// TwinCAT 3 PLC project MAS418_PLC
// ProgramVersion: 3.1.4023.0
// libraries:
//   Tc2_Standard, * (Beckhoff Automation GmbH)
//   Tc2_System, * (Beckhoff Automation GmbH)
//   Tc3_Module, * (Beckhoff Automation GmbH)
// project tree:
//   DUTs/ E_ControlBox.TcDUT, E_Mode.TcDUT, E_Status.TcDUT, ST_Joystick.TcDUT, ST_JoystickInputScaling.TcDUT, ST_Params.TcDUT, ST_Position.TcDUT, ST_PressureSensors.TcDUT, ST_ValveDeadBand.TcDUT
//   Fbs/ FB_ControlBox.TcPOU, FB_Encoder.TcPOU, FB_JoystickInputScaling.TcPOU, FB_RealControlBox_.TcPOU, FB_12bIntToReal.TcPOU, FB_ValveOutput.TcPOU, FB_VirtualControlBox.TcPOU
//   / GlobalTextList.TcGTLO, I_ControlBox.TcIO, I_Crane.TcIO, PlcTask.TcTTO, Visualization Manager.TcVMO (not stored)
//   GVLs/ CONSTANTS.TcGVL, INPUT.TcGVL, OUTPUTS.TcGVL, ScaledInputs.TcGVL, VirtualControlBox.TcGVL, Working.TcGVL
//   POUs/ CraneControl.TcPOU, FU_Scale_IO.TcPOU, MAIN.TcPOU
//   VISUs/ VirtualControlBox.TcVIS
// real-time tasks:
//   TASK PlcTask: cycle T#10ms, priority 20, ADS port 350
// I/O:
//   DEVICE Device 2 (EtherCAT), AmsNetId 5.80.90.242.3.1
//     Term 1 (EK1200) [EK1200-5000 EtherCAT Power supply (2A E-Bus)]
//       Term 10 (EL2008-0015) [EL2008-0015 8Ch. Dig. Output 24V DC, 0.35A, not short-circuit proof]
//       Term 3 (EL9011) [EL9011 End Terminal]
//   DEVICE Device 5 (EtherCAT), AmsNetId 5.80.90.242.6.1
//     Term 12 (EK1100) [EK1100 EtherCAT Coupler (2A E-Bus)]
//       DI1(EL1008) [EL1008 8Ch. Dig. Input 24V, 3ms]
//       DO1(EL2008) [EL2008 8Ch. Dig. Output 24V, 0.5A]
//       AI1(EL3068) [EL3068 8Ch. Ana. Input 0-10V]
//       AI2(EL3068) [EL3068 8Ch. Ana. Input 0-10V]
//       AI3(EL3174) [EL3174 4Ch. Ana. Input +/-10V Diff., +/-20mA SingleEnded, 16 Bit]
//       AI4(EL3255) [EL3255 5Ch. potentiometer measurement with sensor supply]
//       Term 19 (EL4104) [EL4104 4Ch. Ana. Output 0-10V, 16bit]
//       AO1(EL9011) [EL9011 End Terminal]
//     Box 20 (Fraba EtherCAT) [Absolute Rotary Encoder IXARC V01.05]
// variable links:
//   MAS418-PLC Instance <-> Device 5 (EtherCAT)/Box 20 (Fraba EtherCAT)
//     PlcTask Inputs/INPUT.nEncoder <-> Encoder/Position Value
//   MAS418-PLC Instance <-> Device 5 (EtherCAT)/Term 12 (EK1100)/AI1(EL3068)
//     PlcTask Inputs/INPUT.nPC_A <-> AI Standard Channel 4/Value
//     PlcTask Inputs/INPUT.nPC_B <-> AI Standard Channel 3/Value
//     PlcTask Inputs/INPUT.nPR <-> AI Standard Channel 2/Value
//     PlcTask Inputs/INPUT.nPS <-> AI Standard Channel 1/Value
//     PlcTask Inputs/INPUT.nPW_A <-> AI Standard Channel 7/Status
//     PlcTask Inputs/INPUT.nPW_A1 <-> AI Standard Channel 5/Value
//     PlcTask Inputs/INPUT.nPW_B <-> AI Standard Channel 8/Value
//     PlcTask Inputs/INPUT.nPW_B1 <-> AI Standard Channel 6/Value
//   MAS418-PLC Instance <-> Device 5 (EtherCAT)/Term 12 (EK1100)/AI2(EL3068)
//     PlcTask Inputs/INPUT.nPW_D <-> AI Standard Channel 1/Value
//     PlcTask Inputs/INPUT.nQW <-> AI Standard Channel 2/Value
//   MAS418-PLC Instance <-> Device 5 (EtherCAT)/Term 12 (EK1100)/AI4(EL3255)
//     PlcTask Inputs/INPUT.nJoyX <-> AI Standard Channel 2/Value
//     PlcTask Inputs/INPUT.nJoyY <-> AI Standard Channel 3/Value
//     PlcTask Inputs/INPUT.nXc <-> AI Standard Channel 1/Value
//   MAS418-PLC Instance <-> Device 5 (EtherCAT)/Term 12 (EK1100)/DI1(EL1008)
//     PlcTask Inputs/INPUT.bAuto <-> Channel 2/Input
//     PlcTask Inputs/INPUT.bJoystick <-> Channel 5/Input
//     PlcTask Inputs/INPUT.bManual <-> Channel 1/Input
//     PlcTask Inputs/INPUT.bStart <-> Channel 3/Input
//     PlcTask Inputs/INPUT.bStop <-> Channel 4/Input
//   MAS418-PLC Instance <-> Device 5 (EtherCAT)/Term 12 (EK1100)/DO1(EL2008)
//     PlcTask Outputs/OUTPUTS.bEnableCylValve <-> Channel 4/Output
//     PlcTask Outputs/OUTPUTS.bEnableWinchValve <-> Channel 3/Output
//     PlcTask Outputs/OUTPUTS.bGreenLed <-> Channel 1/Output
//     PlcTask Outputs/OUTPUTS.bRedLed <-> Channel 2/Output
//   MAS418-PLC Instance <-> Device 5 (EtherCAT)/Term 12 (EK1100)/Term 19 (EL4104)
//     PlcTask Outputs/OUTPUTS.nCylValveOut <-> AO Output Channel 2/Analog output
//     PlcTask Outputs/OUTPUTS.nWinchValveOut <-> AO Output Channel 1/Analog output

CONFIGURATION MAS418_PLC
    RESOURCE PLC ON TwinCAT3
        TASK PlcTask(INTERVAL := T#10ms, PRIORITY := 20);
        PROGRAM MAIN WITH PlcTask : MAIN;
    END_RESOURCE
END_CONFIGURATION

// ---- DUTs/E_ControlBox.TcDUT
{attribute 'qualified_only'}
{attribute 'strict'}
TYPE E_ControlBox :
(
	VirtualControlBox,
	RealControlBox
);
END_TYPE

// ---- DUTs/E_Mode.TcDUT
{attribute 'qualified_only'}
{attribute 'strict'}
TYPE E_Mode :
(
	AUTO := 0,
	OFF := 1,
	MANUAL := 2
);
END_TYPE

// ---- DUTs/E_Status.TcDUT
{attribute 'qualified_only'}
{attribute 'strict'}
TYPE E_Status :
(
	NotReady,
	Ready,
	Starting,
	Running,
	Stopping,
	Fault,
	Joystick
);
END_TYPE

// ---- DUTs/ST_Joystick.TcDUT
TYPE ST_Joystick :
STRUCT
	X : LREAL;
	Y : LREAL;
	Topswitch : BOOL;
END_STRUCT
END_TYPE

// ---- DUTs/ST_JoystickInputScaling.TcDUT
TYPE ST_JoystickInputScaling :
STRUCT
	
    fMaxInputValue : LREAL := 20509.0;
    fMinInputValue : LREAL := 11787.0;
    fNeutralInputValue : LREAL := 16175;
    fNeutralDeadband : LREAL := 50.0;
    fMaxOutputValue : LREAL := 1.0;
    fMinOutputValue : LREAL := -1.0;
    fNeutralOutputValue : LREAL := 0.0;

END_STRUCT
END_TYPE

// ---- DUTs/ST_Params.TcDUT
TYPE ST_Params :
STRUCT
	fEncoderOffset : LREAL;
END_STRUCT
END_TYPE

// ---- DUTs/ST_Position.TcDUT
TYPE ST_Position :
STRUCT
	winch : REAL;
	cylinder : REAL;
END_STRUCT
END_TYPE

// ---- DUTs/ST_PressureSensors.TcDUT
TYPE ST_PressureSensors :
STRUCT
	SupplyPres : REAL;
	ReturnPres : REAL;
	CylPistSide : REAL;
	CylRodSide : REAL;
	WinchInlet : REAL;
	WinchInlet2 : REAL;
	WinchOutlet : REAL;
	WinchOutlet2 : REAL;
	WinchDrain : REAL;
END_STRUCT
END_TYPE

// ---- DUTs/ST_ValveDeadBand.TcDUT
TYPE ST_ValveDeadBand :
STRUCT
	
    fPosMax : LREAL := 29490.0;
    fPosMin : LREAL  := 20950.0;
    fNegMin : LREAL  := 18250.0;
    fNegMax : LREAL  := 9830.0;

END_STRUCT
END_TYPE

// ---- GVLs/CONSTANTS.TcGVL
{attribute 'qualified_only'}
VAR_GLOBAL
	fDrumD : REAL := 0.475; //m
	fGearRatio : REAL := 1/20;
	//fMdisplacement	: REAL := 
	
END_VAR

// ---- GVLs/INPUT.TcGVL
{attribute 'qualified_only'}
VAR_GLOBAL
//	nJoyXRaw : INT;
//	nJoyYRaw : INT;
//	bJoySW 	: BOOL;
	
	//Digital
	bManual AT %I*: BOOL;
	bAuto AT %I*: BOOL;
	bStart AT %I*: BOOL;
	bStop AT %I*: BOOL;
	bJoystick AT %I*: BOOL;
	
	//Encoder
	nEncoder AT %I*: UDINT;
	
	//Analog Flow/pressure
	nPS AT %I*: INT;
	nPR AT %I*: INT;
	nPC_B  AT %I*: INT;
	nPC_A  AT %I*: INT;
	nPW_A1  AT %I*: INT;
	nPW_B1 AT %I*: INT;
	nPW_A AT %I*: INT;
	nPW_B AT %I*: INT;
	nPW_D AT %I*: INT;
	nQW AT %I*: INT;
	
	//Analog 
	nXc AT %I*: INT;
	//nJoy
	nJoyX AT %I*: INT;
	nJoyY AT %I*: INT;
	
//	fCylinderPositionSensor : REAL;
//	fWinchEncodder : REAL;
//	stPressureSensors : ST_PressureSensors;
//	WinchInletFlow : REAL;
	//I
END_VAR

// ---- GVLs/OUTPUTS.TcGVL
{attribute 'qualified_only'}
VAR_GLOBAL
	//bLightRed : BOOL := FALSE;
	//bLightGreen : BOOL := FALSE;
	//CylinderValve : REAL := 0; //initial value
	//WinchValve : REAL := 0; //initial value
	
	//Digital
	bGreenLed AT %Q*: BOOL;
	bRedLed AT %Q*: BOOL;
	bEnableWinchValve AT %Q*: BOOL;
	bEnableCylValve AT %Q*: BOOL;
	
	//Analog
	nWinchValveOut AT %Q*: INT;
	nCylValveOut AT %Q*: INT;
	
END_VAR

// ---- GVLs/ScaledInputs.TcGVL
{attribute 'qualified_only'}
VAR_GLOBAL
	stJoystick : ST_Joystick;
	
	//Analog Flow/pressure
	fPS : LREAL;
	fPR : LREAL;
	fPC_B : LREAL;
	fPC_A : LREAL;
	fPW_A1 : LREAL;
	fPW_B1 : LREAL;
	fPW_A : LREAL;
	fPW_B : LREAL;
	fPW_D : LREAL;
	fQW : LREAL;
	fXc: LREAL;
	
	fEncoder : LREAL;
	
	
	
END_VAR

// ---- GVLs/VirtualControlBox.TcGVL
{attribute 'qualified_only'}
VAR_GLOBAL
	bSTOP : BOOL := FALSE;
	bSTART : BOOL := FALSE;
	//bLightRed : BOOL := FALSE;
	//bLightGreen : BOOL := FALSE;
	bAuto : BOOL;
	bManual : BOOL;
	stJOY : ST_Joystick;
	//eMode : E_Mode;// := E_Mode.OFF;
	//strMode : STRING;
	//strStatus : STRING;
	//eStatus : E_Status;// := E_Status.NotReady;
	//eMode : E_Mode;// := E_Mode.OFF;
END_VAR

// ---- GVLs/Working.TcGVL
{attribute 'qualified_only'}
VAR_GLOBAL
	eMode : E_Mode;
	eStatus : E_Status := E_Status.NotReady; //Initial status
	strMode : STRING;
	strStatus : STRING;
END_VAR

// ---- I_ControlBox.TcIO
INTERFACE I_ControlBox

METHOD Joystick
VAR_INPUT
	//stJoystick : ST_Joystick;
END_VAR
VAR_OUTPUT
	stJoystick : ST_Joystick;
END_VAR
END_METHOD

METHOD Mode
VAR_INPUT
	//bAuto : BOOL;
	//bManual : BOOL;
	//eMode	: E_Mode; //should I read this value Directly from the VirtualControlBox?
END_VAR
VAR_OUTPUT
	eMode : E_Mode;
END_VAR
END_METHOD

METHOD Status
VAR_INPUT
	//eMode	: E_Mode;
	//bStart	: BOOL;
	//bStop	: BOOL;
END_VAR
VAR_OUTPUT
	//eStatus : E_Status := E_Status.NotReady;
END_VAR
END_METHOD

END_INTERFACE

// ---- I_Crane.TcIO
INTERFACE I_Crane

METHOD ControlValveOutput
VAR_INPUT
END_VAR
END_METHOD

METHOD FLOW : REAL
VAR_INPUT
END_VAR
END_METHOD

METHOD Position : ST_Position
VAR_INPUT
END_VAR
END_METHOD

METHOD Pressure : REAL
VAR_INPUT
END_VAR
END_METHOD

END_INTERFACE

// ---- POUs/MAIN.TcPOU
PROGRAM MAIN
VAR
END_VAR

CraneControl();

END_PROGRAM

// ---- POUs/CraneControl.TcPOU
PROGRAM CraneControl
VAR
	fbControlBox : FB_ControlBox;
	fbScaleOutputs : FB_ValveOutput;
	stValveDeadband : ST_ValveDeadBand;
	//eMode : E_Mode;
	eStatus : E_Status;
	bEnableCylinder : BOOL;
	bEnableWinch	: BOOL;
END_VAR

fbControlBox(eControlBox := E_ControlBox.VirtualControlBox); // set to true to use real controlbox

FU_Scale_IO();

eStatus:=Working.eStatus;
//Control Lights
IF eStatus = E_Status.Running THEN
	OUTPUTS.bGreenLed := TRUE;
	bEnableCylinder := TRUE;
	IF ScaledInputs.stJoystick.Topswitch THEN
		bEnableWinch := TRUE;
	ELSE
		bEnableWinch := FALSE;
	END_IF
ELSE
	OUTPUTS.bGreenLed := FALSE;
	bEnableCylinder := FALSE;
	bEnableWinch := FALSE;
END_IF

IF eStatus = E_Status.Stopping OR eStatus = E_Status.Fault THEN
	OUTPUTS.bRedLed := TRUE;
ELSE
	OUTPUTS.bRedLed := FALSE;
END_IF


//Outputs
fbScaleOutputs(bEnable:=bEnableCylinder, 
			bDeadBandCompOn:=TRUE, 
			stValveDeadBand:=stValveDeadband, 
			fNormalizedInput:=ScaledInputs.stJoystick.X, 
			bEnableValveOutput=>OUTPUTS.bEnableCylValve, 
			nOutput=>OUTPUTS.nCylValveOut);
			
fbScaleOutputs(bEnable:=bEnableWinch, 
			bDeadBandCompOn:=TRUE, 
			stValveDeadBand:=stValveDeadband, 
			fNormalizedInput:=ScaledInputs.stJoystick.Y, 
			bEnableValveOutput=>OUTPUTS.bEnableWinchValve, 
			nOutput=>OUTPUTS.nWinchValveOut);

END_PROGRAM

// ---- Fbs/FB_ControlBox.TcPOU
FUNCTION_BLOCK FB_ControlBox
VAR_INPUT
	eControlBox : E_ControlBox;
END_VAR
VAR
	fbVirtualControlBox : FB_VirtualControlBox;
	fbRealControlBox : FB_RealControlBox_;
	fbControlBox : I_ControlBox := fbVirtualControlBox; //Initial value
END_VAR

CASE eControlBox OF
	E_ControlBox.RealControlBox:
		fbControlBox := fbRealControlBox;
		
	E_ControlBox.VirtualControlBox:
		fbControlBox := fbVirtualControlBox;
END_CASE

fbControlBox.Mode();
fbControlBox.Status();
fbControlBox.Joystick();

END_FUNCTION_BLOCK

// ---- Fbs/FB_VirtualControlBox.TcPOU
FUNCTION_BLOCK FB_VirtualControlBox IMPLEMENTS I_ControlBox
VAR_INPUT
END_VAR
VAR_OUTPUT
END_VAR
VAR
END_VAR

//fbControlBox.Mode(
//	bAuto := VirtualControlBox.bAuto, 
//	bManual := VirtualControlBox.bManual,
//	eMode => VirtualControlBox.eMode
//);

//fbControlBox.Status(
//	eMode := VirtualControlBox.eMode,
//	bStart := VirtualControlBox.bSTART,
//	bStop := VirtualControlBox.bSTOP,
//	eStatus => VirtualControlBox.eStatus
//	);

{warning 'add method implementation '}
METHOD Joystick
VAR_INPUT
	//stJoystick	: ST_Joystick;
END_VAR
VAR_OUTPUT
	stJoystick : ST_Joystick;
END_VAR
VAR
	
END_VAR
ScaledInputs.stJoystick := VirtualControlBox.stJOY;

ScaledInputs.stJoystick.Topswitch := VirtualControlBox.stJOY.Topswitch;
//ScaledInputs.stJoystick := stJoystick;
END_METHOD

{warning 'add method implementation '}
METHOD Mode
VAR_INPUT
	//bAuto : BOOL;
	//bManual : BOOL;
	//eMode	: E_Mode; //should I read this value Directly from the VirtualControlBox?
END_VAR
VAR_OUTPUT
	eMode : E_Mode;
END_VAR

VAR
	//eMode : E_Mode;
	bAuto : BOOL;
	bManual : BOOL;
END_VAR
//eMode := VirtualControlBox.eMode;
//OUTPUTS.eMode := eMode;

bAuto := VirtualControlBox.bAuto;
bManual := VirtualControlBox.bManual;


IF bAuto AND NOT bManual THEN
	eMode := E_Mode.AUTO;
	Working.strMode := 'AUTO';
ELSIF bManual AND NOT bAuto THEN
	eMode := E_Mode.MANUAL;
	Working.strMode := 'MANUAL';
ELSE
	eMode := E_Mode.OFF;
	Working.strMode := 'OFF';
END_IF

Working.eMode := eMode;
END_METHOD

{warning 'add method implementation '}
METHOD Status
VAR_INPUT
	//eMode	: E_Mode;
	//bStart	: BOOL;
	//bStop	: BOOL;
END_VAR
VAR_OUTPUT
	//eStatus : E_Status := E_Status.NotReady;
END_VAR
VAR
	eStatus : E_Status;
	eMode : E_Mode;
END_VAR
eMode := Working.eMode;
eStatus := Working.eStatus;
CASE eStatus OF
	E_Status.NotReady:
		Working.strStatus := 'NotReady';
		IF eMode <> E_Mode.OFF THEN
			eStatus := E_Status.Ready;
		END_IF
	
	E_Status.Ready:
		Working.strStatus := 'Ready';
		IF eMode = E_Mode.OFF THEN
			eStatus := E_Status.NotReady;
		ELSIF VirtualControlBox.bStart THEN
			eStatus := E_Status.Starting;
		END_IF
		
	E_Status.Starting:
		Working.strStatus := 'Starting';
		IF VirtualControlBox.bStart AND NOT VirtualControlBox.bStop THEN //Add more start conditions?
			eStatus := E_Status.Running;	
		ELSE
			eStatus := E_Status.Ready;
		END_IF
		
	E_Status.Running:	
		Working.strStatus := 'Running';
		IF VirtualControlBox.bStop THEN
			eStatus := E_Status.Stopping;
		ELSIF eMode = E_Mode.AUTO THEN
			IF NOT VirtualControlBox.bStart THEN // ADD Clock signal
				eStatus := E_Status.Stopping;
			END_IF	
		END_IF
		
	E_Status.Stopping:
		Working.strStatus := 'Stopping';
		//Add stop condition
		eStatus := E_Status.NotReady;
		
	E_Status.Fault:
		Working.strStatus := 'Fault';				
END_CASE

Working.eStatus := eStatus;

////Control Lights
//IF eStatus = E_Status.Running THEN
//	OUTPUTS.bGreenLed := TRUE;
//	OUTPUTS.bEnableCylValve := TRUE;
//	IF ScaledInputs.stJoystick.Topswitch THEN
//		OUTPUTS.bEnableWinchValve := TRUE;
//	ELSE
//		OUTPUTS.bEnableWinchValve := FALSE;
//	END_IF
//ELSE
//	OUTPUTS.bGreenLed := FALSE;
//	OUTPUTS.bEnableCylValve := FALSE;
//	OUTPUTS.bEnableWinchValve := FALSE;
//END_IF

//IF eStatus = E_Status.Stopping OR eStatus = E_Status.Fault THEN
//	OUTPUTS.bRedLed := TRUE;
//ELSE
//	OUTPUTS.bRedLed := FALSE;
//END_IF
END_METHOD

END_FUNCTION_BLOCK

// ---- Fbs/FB_RealControlBox_.TcPOU
FUNCTION_BLOCK FB_RealControlBox_ IMPLEMENTS I_ControlBox
VAR_INPUT
END_VAR
VAR_OUTPUT
END_VAR
VAR
END_VAR

{warning 'add method implementation '}
METHOD Joystick
VAR_OUTPUT
	stJoystick	: ST_Joystick;
END_VAR
VAR
	fbJoystickInputScaling : FB_JoystickInputScaling;
	stJoystickInputScaling : ST_JoystickInputScaling;
	//nXInput: INT;
	//nYInput: INT;
END_VAR
//stJoystick := VirtualControlBox.stJOY;
fbJoystickInputScaling(bEnable:=TRUE, 
		nRawInput:=INPUT.nJoyX, 
		stJoystickInputScaling:=stJoystickInputScaling, 
		fNormalizedOutput => ScaledInputs.stJoystick.X);

		
fbJoystickInputScaling(bEnable:=TRUE, 
		nRawInput:=INPUT.nJoyY, 
		stJoystickInputScaling:=stJoystickInputScaling, 
		fNormalizedOutput => ScaledInputs.stJoystick.Y);

ScaledInputs.stJoystick.Topswitch := INPUT.bJoystick;
END_METHOD

{warning 'add method implementation '}
METHOD Mode
VAR_OUTPUT
	eMode	: E_Mode;
END_VAR
VAR
	//eMode : E_Mode;
	bAuto : BOOL;
	bManual : BOOL;
END_VAR
//eMode := VirtualControlBox.eMode;
//OUTPUTS.eMode := eMode;

bAuto := INPUT.bAuto;
bManual := INPUT.bManual;


IF bAuto AND NOT bManual THEN
	eMode := E_Mode.AUTO;
	Working.strMode := 'AUTO';
ELSIF bManual AND NOT bAuto THEN
	eMode := E_Mode.MANUAL;
	Working.strMode := 'MANUAL';
ELSE
	eMode := E_Mode.OFF;
	Working.strMode := 'OFF';
END_IF

Working.eMode := eMode;
END_METHOD

{warning 'add method implementation '}
METHOD Status
VAR
	eStatus : E_Status;
	eMode : E_Mode;
END_VAR
eMode := Working.eMode;
eStatus := Working.eStatus;
CASE eStatus OF
	E_Status.NotReady:
		Working.strStatus := 'NotReady';
		IF eMode <> E_Mode.OFF THEN
			eStatus := E_Status.Ready;
		END_IF
	
	E_Status.Ready:
		Working.strStatus := 'Ready';
		IF eMode = E_Mode.OFF THEN
			eStatus := E_Status.NotReady;
		ELSIF INPUT.bStart THEN
			eStatus := E_Status.Starting;
		END_IF
		
	E_Status.Starting:
		Working.strStatus := 'Starting';
		IF INPUT.bStart AND NOT INPUT.bStop THEN //Add more start conditions?
			eStatus := E_Status.Running;	
		ELSE
			eStatus := E_Status.Ready;
		END_IF
		
	E_Status.Running:	
		Working.strStatus := 'Running';
		IF INPUT.bStop THEN
			eStatus := E_Status.Stopping;
		ELSIF eMode = E_Mode.AUTO THEN
			IF NOT INPUT.bStart THEN // ADD Clock signal
				eStatus := E_Status.Stopping;
			END_IF	
		END_IF
		
	E_Status.Stopping:
		Working.strStatus := 'Stopping';
		//Add stop condition
		eStatus := E_Status.NotReady;
		
	E_Status.Fault:
		Working.strStatus := 'Fault';				
END_CASE

Working.eStatus := eStatus;

//Control Lights
//IF eStatus = E_Status.Running THEN
//	OUTPUTS.bGreenLed := TRUE;
//	OUTPUTS.bEnableCylValve := TRUE;
//	IF ScaledInputs.stJoystick.Topswitch THEN
//		OUTPUTS.bEnableWinchValve := TRUE;
//	ELSE
//		OUTPUTS.bEnableWinchValve := FALSE;
//	END_IF
//ELSE
//	OUTPUTS.bGreenLed := FALSE;
//	OUTPUTS.bEnableCylValve := FALSE;
//	OUTPUTS.bEnableWinchValve := FALSE;
//END_IF

//IF eStatus = E_Status.Stopping OR eStatus = E_Status.Fault THEN
//	OUTPUTS.bRedLed := TRUE;
//ELSE
//	OUTPUTS.bRedLed := FALSE;
//END_IF
END_METHOD

END_FUNCTION_BLOCK

// ---- Fbs/FB_JoystickInputScaling.TcPOU
FUNCTION_BLOCK FB_JoystickInputScaling
VAR_INPUT
	bEnable 	: BOOL;
	nRawInput	: INT;
	stJoystickInputScaling	: ST_JoystickInputScaling;
END_VAR
VAR_OUTPUT
	fNormalizedOutput	: LREAL;
END_VAR
VAR
	fRawInput	: LREAL;
	fTempInput	: LREAL;
	fTempOutput	: LREAL;
END_VAR

fRawInput := INT_TO_LREAL(nRawInput);

fTempInput := fRawInput - stJoystickInputScaling.fNeutralInputValue;

IF fTempInput > stJoystickInputScaling.fNeutralDeadband THEN
	fTempOutput := fTempInput/(stJoystickInputScaling.fMaxInputValue - stJoystickInputScaling.fNeutralInputValue);
ELSIF fTempInput < stJoystickInputScaling.fNeutralDeadband THEN
	fTempOutput := fTempInput/(stJoystickInputScaling.fNeutralInputValue - stJoystickInputScaling.fMinInputValue);
ELSE 
	fTempOutput := 0.0;
END_IF

IF NOT(bEnable) THEN
	fNormalizedOutput := 0.0;
ELSE
	fNormalizedOutput := LIMIT(stJoystickInputScaling.fMinOutputValue, fTempOutput, stJoystickInputScaling.fMaxOutputValue);
END_IF

END_FUNCTION_BLOCK

// ---- Fbs/FB_ValveOutput.TcPOU
FUNCTION_BLOCK FB_ValveOutput
VAR_INPUT
	bEnable	: BOOL;
	bDeadBandCompOn	:BOOL;
	stValveDeadBand	: ST_ValveDeadBand;
	fNormalizedInput	: LREAL;
END_VAR
VAR_OUTPUT
	bEnableValveOutput	: BOOL;
	nOutput 			: INT;
END_VAR
VAR
	nOffset		: INT := 19660;
	nMaxValue	: INT := 29490;
	nMinValue	: INT := 9830;
	nTempOutput	: INT;
END_VAR

IF bDeadBandCompOn THEN
	IF fNormalizedInput > 0.0 THEN
		nTempOutput := LREAL_TO_INT(ABS(fNormalizedInput*(stValveDeadBand.fPosMax - stValveDeadBand.fPosMin) + stValveDeadBand.fPosMin));
	ELSIF fNormalizedInput < 0.0 THEN
		nTempOutput := LREAL_TO_INT(ABS(fNormalizedInput*(stValveDeadBand.fNegMax - stValveDeadBand.fNegMin) - stValveDeadBand.fNegMin));
	ELSE
		nTempOutput := nOffset;
	END_IF
ELSE
	IF fNormalizedInput > 0.0 THEN
		nTempOutput := LREAL_TO_INT(ABS(fNormalizedInput*(32767.0 - 19660.0) + 19660.0));
	ELSIF fNormalizedInput < 0.0 THEN
		nTempOutput := LREAL_TO_INT(ABS(fNormalizedInput*(0.0 - 19660.0) + 19660.0));
	ELSE 
		nTempOutput := nOffset;
	END_IF
END_IF

IF bEnable THEN
	nOutput := LIMIT(nMinValue, nTempOutput, nMaxValue);
	bEnableValveOutput := TRUE;
ELSE
	nOutput := nOffset;
	bEnableValveOutput := FALSE;
END_IF

END_FUNCTION_BLOCK

// ---- POUs/FU_Scale_IO.TcPOU
FUNCTION FU_Scale_IO : BOOL
VAR_INPUT
END_VAR
VAR
	fbScale : FB_12bIntToReal;
END_VAR

fbScale(nInput:=INPUT.nXc, fMin:=0, fMax:=0.5, fOutput => ScaledInputs.fXc);
fbScale(nInput:=INPUT.nPS, fMin:=0, fMax:=400, fOutput => ScaledInputs.fPS);
fbScale(nInput:=INPUT.nPR, fMin:=0, fMax:=40, fOutput => ScaledInputs.fPR);
fbScale(nInput:=INPUT.nPC_A, fMin:=0, fMax:=400, fOutput => ScaledInputs.fPC_A);
fbScale(nInput:=INPUT.nPC_B, fMin:=0, fMax:=400, fOutput => ScaledInputs.fPC_B);
fbScale(nInput:=INPUT.nPW_A, fMin:=0, fMax:=400, fOutput => ScaledInputs.fPW_A);
fbScale(nInput:=INPUT.nPW_A1, fMin:=0, fMax:=400, fOutput => ScaledInputs.fPW_A1);
fbScale(nInput:=INPUT.nPW_B, fMin:=0, fMax:=400, fOutput => ScaledInputs.fPW_B);
fbScale(nInput:=INPUT.nPW_B1, fMin:=0, fMax:=400, fOutput => ScaledInputs.fPW_B1);
fbScale(nInput:=INPUT.nPW_D, fMin:=0, fMax:=40, fOutput => ScaledInputs.fPW_D);
fbScale(nInput:=INPUT.nQW, fMin:=-150, fMax:=150, fOutput => ScaledInputs.fQw);

END_FUNCTION

// ---- Fbs/FB_12bIntToReal.TcPOU
FUNCTION_BLOCK FB_12bIntToReal
VAR_INPUT
	nInput : INT;
	fMin	: LREAL;
	fMax	: LREAL;
	
END_VAR
VAR_OUTPUT
	fOutput : LREAL;
END_VAR
VAR
	fRange : LREAL;
	fScale : LREAL;
	//fResolution12Bit : LREAL := 4095;
	fResolution12Bit : LREAL := 32767;
END_VAR

//fRange := INT_TO_LREAL(iMax-iMin);
fRange := fMax-fMin;
fScale := fRange/fResolution12Bit;
fOutput := INT_TO_LREAL(nInput) * fScale + fMin;

END_FUNCTION_BLOCK

// ---- Fbs/FB_Encoder.TcPOU
FUNCTION_BLOCK FB_Encoder
VAR_INPUT
	nRawInput : UDINT;
	stParam	:	ST_Parameters;
END_VAR
VAR_OUTPUT
	fPosition : LREAL;
END_VAR
VAR PERSISTENT
	nRounds	: DINT;
	nRawLast : DINT;
END_VAR
VAR
	nInput : DINT;
	nTempInputDiff : DINT;
	nCount	: DINT;
	nMaxValue30bit	: DINT := 1073741823;
	nThreshold30bit	: DINT := nMaxValue30bit/2;
	fScale16bit : LREAL := 360.0/65535.0;
	fTempPosition	:LREAL;
END_VAR

// Convert to DINT
nInput := UDINT_TO_DINT(nRawInput);

nTempInputDiff := nInput - nRawLast;
IF(nTempInputDiff > nThreshold30bit) THEN
	nRounds := nRounds -1;
END_IF
IF (nTempInputDiff < -nThreshold30bit) THEN
	nRounds := nRounds + 1;
END_IF

//Count Encoder Rounds
nCount := nInput + nRounds*nMaxValue30bit;

//Position output
fPosition := DINT_TO_LREAL(nCount)*fScale16bit - stParam.fEncoderOffset;

nRawLast := nInput;

END_FUNCTION_BLOCK

// ---- GlobalTextList.TcGTLO
TEXTLIST GlobalTextList
  610 = '"JOY\\nTopSwitch"'
  786 = '%s'
  277 = 'AUTO'
  56 = 'Auto'
  308 = 'ControlBox'
  504 = 'JOYTopSwitch'
  507 = 'JOY\\nTopSwitch'
  846 = 'JOY_TopSwitch'
  460 = 'JOY_X'
  698 = 'JOY_Y'
  914 = 'MANUAL'
  767 = 'Manuel'
  731 = 'Mode'
  179 = 'Mode Selector'
  157 = 'Mode:'
  874 = 'OFF'
  683 = 'Off'
  787 = 'Selector switch'
  113 = 'START'
  214 = 'Status:'
  682 = 'STOP'
END_TEXTLIST

// ---- VISUs/VirtualControlBox.TcVIS
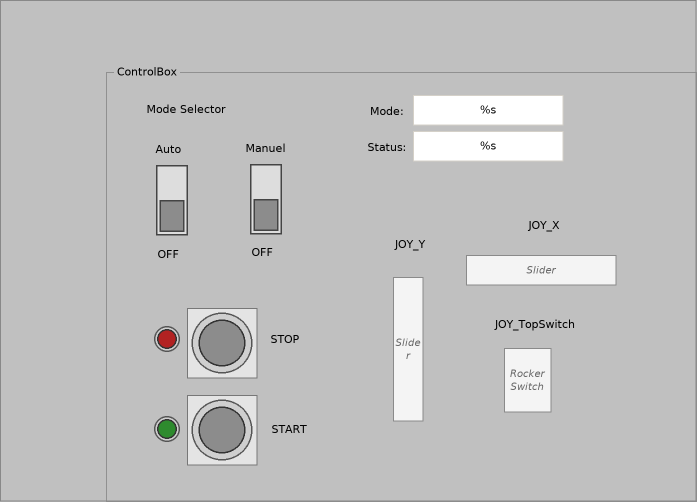
VISUALIZATION VirtualControlBox  // 697x502
    GroupBox (106,64 591x438), "ControlBox"
        PushSwitch (81,244 70x70), variable: VirtualControlBox.bSTOP, behaviour: TOGGLE, style: Switch-PushSwitch-Gray
        PushSwitch (81,331 70x70), variable: VirtualControlBox.bSTART, behaviour: TOGGLE, style: Switch-PushSwitch-Gray
        Slider (360,191 150x30), variable: VirtualControlBox.stJOY.X, scale -1..1
        Slider (287,213 30x144), variable: VirtualControlBox.stJOY.Y, scale -1..1
        RockerSwitch (398,284 47x64), variable: VirtualControlBox.stJOY.Topswitch, behaviour: TOGGLE, style: Switch-RockerSwitch-Gray
        Textfield (307,31 150x30), "%s", text variable: Working.strMode
        Label (378,247 102x27), "JOY_TopSwitch"
        Label (387,148 102x27), "JOY_X"
        Label (253,167 102x27), "JOY_Y"
        Label (233,34 96x27), "Mode:"
        Label (230,70 102x27), "Status:"
        Label (29,32 102x27), "Mode Selector"
        Label (132,352 102x27), "START"
        Label (128,262 102x27), "STOP"
        Lamp1 (46,260 30x30), variable: OUTPUTS.bRedLed, style: Lamp-Lamp1-Red
        Lamp1 (46,350 30x30), variable: OUTPUTS.bGreenLed, style: Lamp-Lamp1-Green
        DipSwitch (31,101 70x70), variable: VirtualControlBox.bAuto, behaviour: TOGGLE, style: Switch-DipSwitch-Gray
        DipSwitch (125,100 70x70), variable: VirtualControlBox.bManual, behaviour: TOGGLE, style: Switch-DipSwitch-Gray
        Label (18,71 89x29), "Auto"
        Label (115,70 89x29), "Manuel"
        Label (18,176 89x29), "OFF"
        Label (112,174 89x29), "OFF"
    Textfield (413,131 150x30), "%s", text variable: Working.strStatus
END_VISUALIZATION
